PROGRAM MAIN
VAR
	fbStateMachine : FB_StateMachine;
END_VAR

fbStateMachine();

END_PROGRAM

(* stored: Version 1.1.0.1, ProductVersion 3.1.4024.12
   POU MAIN: Id {89cf6417-631f-46b9-9ac5-03ab9c62d2d0}, SpecialFunc None *)
